Universal Robots PolyScope program: ad_lab_exe_4_1_63.urp

Program ad_lab_exe_4_1_63 (createdIn=3.2.19293 lastSavedIn=3.2.19293 directory=/programs installation=default robotSerialNumber=2015351391)
Calibrated DH parameters: a=[0.000352, -0.161198, -0.373486, 0.00005, 0.000049, 0]; d=[0.089268, 352.477598, -320.08558, -32.281492, 0.094939, 0.082518]; alpha=[1.570728, 0.001116, -0.003686, 1.571189, -1.570572, 0]; deltaTheta=[-0.000012, 1.181849, -1.491165, 0.309495, -0.000007, 0.000025]
Robot Program (runOnlyOnce=false motionType=MoveJ speed=1.047198 acceleration=1.396263 recalculateMotions=false)
  Folder 文件夹
    tcp1 := p[0,0,0.2,0,0,0]
    tcp2 := p[0.2,0,0.05,0,d2r(90),0]
    Script: set_tcp(tcp1)
    Script: set_tcp(tcp2)
